(* CODESYS project SNDLTN_JSON.library
   Description: Library to convert and handle JSON data.
   Company: Sandolution
   Version: 1.2.200525
   Title: SNDLTN_JSON
   Author: S. Verbeek

Project tree, tasks and I/O mapping:
  libraries: StringUtils, * (System)
  Constants/
    global variables JSON_Properties
    global variables JSON_Constants
  Enums/
    data type JSON_eConversionType
    data type JSON_eError
  Function Blocks/
    function block JSON_Parser [ST]
    function block JSON_GetSingleValue [ST]
    function block JSON_GetMultiValue [ST]
  Functions/
  Structs/
  Variables/
  program ChangeLog [ST]
*)

// Enums/JSON_eConversionType
{attribute 'qualified_only'}
TYPE JSON_eConversionType :
(
	None := 0,				//NO CONVERSION
	Boolean,				//BOOL
	Integer,				//INT
	UnsignedInteger,		//UINT
	DoubleInteger,			//DINT
	UnsignedDoubleInteger,	//UDINT
	FloatingPoint,			//REAL
	DateAndTime,			//DT
	TimeOfDay				//TOD
);
END_TYPE

// Enums/JSON_eError
{attribute 'qualified_only'}
TYPE JSON_eError :
(
	NoError 				:= 0,
	//3000-3999 : JSON ERRORS
	PropertiesArrayToSmall 	:= 3000,	//JSON Parser output array to small
	PropertySizeToSmall 	:= 3001		//JSON Size to small
);
END_TYPE

// Constants/JSON_Properties
{attribute 'qualified_only'}
VAR_GLOBAL CONSTANT
	uiJSONMaxInputSize			:UINT := 4096;
	uiJSONMaxProperties			:UINT := 128;
	uiJSONMaxPropertySize		:UINT := 256;
	uiJSONMaxInputMultiValue	:UINT := 32;

END_VAR

// Constants/JSON_Constants
{attribute 'qualified_only'}
{attribute 'conditionalshow'}
VAR_GLOBAL
	sLineBreak					:STRING(1) := '$N';
	sColom						:STRING(3) := ' : ';
	sComma						:STRING(1) := ',';
	sQuotationMark				:STRING(1) := '"';
	sEnumerationBegin			:STRING(1) := '[';
	sEnumerationEnd				:STRING(1) := ']';
	sAccoladeBegin				:STRING(1) := '{';
	sAccoladeEnd				:STRING(1) := '}';
END_VAR

// Function Blocks/JSON_Parser
{attribute 'conditionalshow_all_locals'}
FUNCTION_BLOCK JSON_Parser
VAR_INPUT
	xResetError				:BOOL;
	sContent				:STRING(JSON_Properties.uiJSONMaxInputSize);
END_VAR
VAR_OUTPUT
	xError					:BOOL;
	eErrorID				:JSON_eError;
	
	//Double array: property/value
	asProperties			:ARRAY[0..1,0..JSON_Properties.uiJSONMaxProperties] OF STRING (JSON_Properties.uiJSONMaxPropertySize);
	uiPropertyCount			:UINT;
	xEnumerationPresent		:BOOL;	//Data contains one or more enumerations of multiple elements
	uiEnumerationIndex		:UINT;	//Start of FIRST enumeration
END_VAR
VAR
	//Store input
	sContent_int			:STRING(JSON_Properties.uiJSONMaxInputSize);
	
	//Input
	psContent				:POINTER TO STRING(JSON_Properties.uiJSONMaxInputSize);
	
	//Get total property line
	sProperty				:STRING(JSON_Properties.uiJSONMaxPropertySize);
	psProperty				:POINTER TO STRING(JSON_Properties.uiJSONMaxPropertySize);
	
	//Search for char (newline / comma / colon)
	sSearch					:STRING(4) := JSON_Constants.sLineBreak;	//Search for line end char
	psSearch				:POINTER TO STRING(4);
	
	//Output
	psProperties			:POINTER TO STRING (JSON_Properties.uiJSONMaxPropertySize);      	
	        
	//Helper            	
	diContentLength			:DINT;	//Length of content
	diPropertyLength		:DINT;	//Length of property
                	
	uiIndex					:UINT;
	
	iPosNewLine				:INT;
	iPosNewLine_Old			:INT;
	
	iPosColom				:INT;
	iPosQuotationMark_Begin	:ARRAY[0..1] OF INT;
	iPosQuotationMark_End	:ARRAY[0..1] OF INT;
	iPosQuotationMark_Loop	:INT;
	iPosComma				:INT;
	
	xOutput_Mem				:BOOL;	//Output written
END_VAR

//Get address and length
psContent := ADR(sContent);
psProperty := ADR(sProperty);
psSearch := ADR(sSearch);
diContentLength := StrLenA(psContent);

//Reset vars
iPosNewLine_Old := -1;	
xOutput_Mem := FALSE;

//Reset outputs
xEnumerationPresent := FALSE;

//Reset error
IF xResetError THEN
	xError := FALSE;
	eErrorID := JSON_eError.NoError;
END_IF

//Loop properties when input changed
IF sContent <> sContent_int THEN
	sContent_int := sContent;

	//Fill output array
	FOR uiIndex := 0 TO JSON_Properties.uiJSONMaxProperties DO
		
		//****************************************************GET PROPERTY FROM STRING (LINE BREAK)
		//Find pos of line break
		sSearch := JSON_Constants.sLineBreak;
		iPosNewLine := StrFindA(psContent, psSearch, TO_UINT(iPosNewLine_Old+1));
		
		IF iPosNewLine > 0 THEN
			
			//Get line at start of string
			IF uiIndex = 0 THEN	
				//Check if content fits the output
				IF (iPosNewLine-1) <= TO_INT(JSON_Properties.uiJSONMaxPropertySize) THEN
					StrMidA(psContent, JSON_Properties.uiJSONMaxInputSize, (iPosNewLine), 1, psProperty, JSON_Properties.uiJSONMaxPropertySize);
				ELSE
					xError := TRUE;
					eErrorID := JSON_eError.PropertySizeToSmall;
					EXIT;
				END_IF
			//Get line after first line
			ELSE	
				//Check if content fits the output
				IF (iPosNewLine-iPosNewLine_Old) <= TO_INT(JSON_Properties.uiJSONMaxPropertySize) THEN
					StrMidA(psContent, JSON_Properties.uiJSONMaxInputSize, (iPosNewLine-iPosNewLine_Old), (iPosNewLine_Old+1), psProperty, JSON_Properties.uiJSONMaxPropertySize);
				ELSE
					xError := TRUE;
					eErrorID := JSON_eError.PropertySizeToSmall;
					EXIT;
				END_IF
			END_IF
			
			//Store var for next find instruction
			iPosNewLine_Old := iPosNewLine;
			
			//****************************************************FIND COLOM IN PROPERTY
			sSearch := JSON_Constants.sColom;
			iPosColom := StrFindA(psProperty, psSearch, 0);
			
			//Column found	
			IF iPosColom > 0 THEN
			
				//****************************************************FIND NAME AND VALUE
				sSearch := JSON_Constants.sQuotationMark;
				//Name
				iPosQuotationMark_Begin[0] := StrFindA(psProperty, psSearch, 0);
				iPosQuotationMark_End[0] := StrFindA(psProperty, psSearch, TO_UINT(iPosQuotationMark_Begin[0]+1));
				
				//Value
				iPosQuotationMark_Begin[1] := StrFindA(psProperty, psSearch, TO_UINT(iPosColom));	//Search after colom
				
				//Start at back of string and work forwards to find latest one, enabling quotation marks in the value
				iPosQuotationMark_End[1] := 0;
				FOR iPosQuotationMark_Loop := TO_INT(StrLenA(psProperty)-1) TO (iPosQuotationMark_Begin[1]+1) BY -1 DO
					iPosQuotationMark_End[1] := StrFindA(psProperty, psSearch, TO_UINT(iPosQuotationMark_Loop));
					//Break if occurance is found
					IF iPosQuotationMark_End[1] <> 0 THEN 
						EXIT; 
					END_IF
				END_FOR
				
				//****************************************************EXTRACT NAME AND VALUE
				//Name
				psProperties := ADR(asProperties[0,uiIndex]);
				IF (iPosQuotationMark_End[0]-iPosQuotationMark_Begin[0]-1) <= TO_INT(JSON_Properties.uiJSONMaxPropertySize) THEN 
					StrMidA(psProperty, JSON_Properties.uiJSONMaxInputSize, (iPosQuotationMark_End[0]-iPosQuotationMark_Begin[0]-1), (iPosQuotationMark_Begin[0]+1), psProperties, JSON_Properties.uiJSONMaxPropertySize);
					StrTrimA(psProperties);	//Remove spaces
				ELSE
					xError := TRUE;
					eErrorID := JSON_eError.PropertySizeToSmall;
					EXIT;
				END_IF
				
				//Value with quotation marks
				psProperties := ADR(asProperties[1,uiIndex]);
				//Check if content fits the output
				IF iPosQuotationMark_Begin[1] > 0 AND iPosQuotationMark_End[1] > 0 THEN
					StrMidA(psProperty, JSON_Properties.uiJSONMaxInputSize, (iPosQuotationMark_End[1]-iPosQuotationMark_Begin[1]-1), (iPosQuotationMark_Begin[1]+1), psProperties, JSON_Properties.uiJSONMaxPropertySize);
					StrTrimA(psProperties);	//Remove spaces			
				
				//Value without quotation marks
				ELSE
					//Search for ending comma
					sSearch := JSON_Constants.sComma;
					iPosComma := StrFindA(psProperty, psSearch, 0);
					diPropertyLength := StrLenA(psProperty);
					//Extract to end of line minus one
					IF iPosComma > 0 THEN
						StrMidA(psProperty, JSON_Properties.uiJSONMaxInputSize, (TO_INT(diPropertyLength)-iPosColom-3-1), (iPosColom+3), psProperties, JSON_Properties.uiJSONMaxPropertySize);	//3> Search argument is ' : "  //1> skip comma
						StrTrimA(psProperties);	//Remove spaces
					//Extract to end of line
					ELSE		
						StrMidA(psProperty, JSON_Properties.uiJSONMaxInputSize, (TO_INT(diPropertyLength)-iPosColom-3), (iPosColom+3), psProperties, JSON_Properties.uiJSONMaxPropertySize);	//3> Search is ' : "
						StrTrimA(psProperties);	//Remove spaces
					END_IF
				END_IF
				
				//Check if there is more data then array size
				IF diContentLength > iPosQuotationMark_End[1] AND uiIndex = JSON_Properties.uiJSONMaxProperties THEN
					xError := TRUE;
					eErrorID := JSON_eError.PropertiesArrayToSmall;
				END_IF
				
				//Check if enumeration is present in array (for e.g. multiple instances of same object)
				//Find function is not used here as value can also be in a value
				IF NOT xEnumerationPresent 
				AND (asProperties[0,uiIndex] = JSON_Constants.sEnumerationBegin OR asProperties[0,uiIndex] = JSON_Constants.sEnumerationEnd
				OR asProperties[1,uiIndex] = JSON_Constants.sEnumerationBegin OR asProperties[1,uiIndex] = JSON_Constants.sEnumerationEnd) THEN
					xEnumerationPresent := TRUE;
					uiEnumerationIndex := uiIndex; 
				END_IF
			
			//No column found > no name+value but different charachter
			ELSE
				//Remove line break
				diPropertyLength := StrLenA(psProperty);
				StrMidA(psProperty, JSON_Properties.uiJSONMaxInputSize, TO_INT(diPropertyLength-1), 1, psProperty, JSON_Properties.uiJSONMaxPropertySize);
				
				//Transfer
				StrTrimA(psProperty);	//Remove spaces
				asProperties[0,uiIndex] := psProperty^;
				asProperties[1,uiIndex] := '';
				
				//Check if enumeration is present in array (for e.g. multiple instances of same object)
				//Find function is not used here as value can also be in a value
				IF NOT xEnumerationPresent 
				AND (asProperties[0,uiIndex] = JSON_Constants.sEnumerationBegin OR asProperties[0,uiIndex] = JSON_Constants.sEnumerationEnd) THEN
					xEnumerationPresent := TRUE;
					uiEnumerationIndex := uiIndex; 
				END_IF
				
			END_IF
			
		//Get latest part of string(should be closing accolade)
		ELSIF iPosNewLine_Old < diContentLength THEN
			IF (TO_INT(diContentLength)-iPosNewLine_Old) <= TO_INT(JSON_Properties.uiJSONMaxPropertySize) THEN
				StrMidA(psContent, JSON_Properties.uiJSONMaxInputSize, (TO_INT(diContentLength)-iPosNewLine_Old-1), iPosNewLine_Old+1, psProperty, JSON_Properties.uiJSONMaxPropertySize);
				StrTrimA(psProperty);	//Remove spaces
			ELSE
				xError := TRUE;
				eErrorID := JSON_eError.PropertySizeToSmall;
				EXIT;
			END_IF
			
			//Transfer data
			asProperties[0,uiIndex] := psProperty^;
			asProperties[1,uiIndex] := '';
			iPosNewLine_Old := TO_INT(diContentLength);
		
		//Closing function
		ELSIF iPosNewLine <= 0 AND iPosNewLine_Old = diContentLength THEN
			
			//Output property count
			IF NOT xOutput_Mem THEN
				xOutput_Mem := TRUE;
				uiPropertyCount := uiIndex;
			END_IF
			
			//Empty array after closing
			IF uiIndex >= uiPropertyCount THEN 
				asProperties[0,uiIndex] := '';
				asProperties[1,uiIndex] := '';
			END_IF
			
		END_IF
		
	END_FOR
END_IF

END_FUNCTION_BLOCK

// Function Blocks/JSON_GetSingleValue
{attribute 'conditionalshow_all_locals'}
FUNCTION_BLOCK JSON_GetSingleValue
VAR_INPUT
	pasProperties		:POINTER TO ARRAY[0..1,0..JSON_Properties.uiJSONMaxProperties] OF STRING(JSON_Properties.uiJSONMaxPropertySize);		//Pointer to output array
	sPropertyName		:STRING(JSON_Properties.uiJSONMaxPropertySize);
	eConversionType		:JSON_eConversionType;
END_VAR
VAR_OUTPUT
	xMatchFound			:BOOL;
	sPropertyValue		:STRING(JSON_Properties.uiJSONMaxPropertySize);		//Always loaded with value
	xPropertyValue		:BOOL;
	iPropertyValue		:INT;
	uiPropertyValue		:UINT;
	diPropertyValue		:DINT;
	udiPropertyValue	:UDINT;
	rPropertyValue		:REAL;
	dtPropertyValue		:DATE_AND_TIME;
	todPropertyValue	:TOD;
END_VAR
VAR
	iIndex				:INT;
	psPropertyValue		:POINTER TO STRING(JSON_Properties.uiJSONMaxPropertySize);
	sSearch				:STRING(8);
	psSearch			:POINTER TO STRING(8);
	iFindResult			:INT;
	
	sReplace			:STRING(1) := '-';
	psReplace			:POINTER TO STRING(4);
	
	sDateTime			:STRING(JSON_Properties.uiJSONMaxPropertySize) := 'DT#';
	psDateTime			:POINTER TO STRING(JSON_Properties.uiJSONMaxPropertySize);
	
	sTimeOfDay			:STRING(JSON_Properties.uiJSONMaxPropertySize) := 'TOD#';
	psTimeOfDay			:POINTER TO STRING(JSON_Properties.uiJSONMaxPropertySize);
	sTimeOfDay_Seconds	:STRING(JSON_Properties.uiJSONMaxPropertySize) := ':00';
	psTimeOfDay_Seconds	:POINTER TO STRING(JSON_Properties.uiJSONMaxPropertySize);
	
	iLengthTOD			:INT;
END_VAR

//Reset values
xMatchFound := FALSE;	//Assume no match is found
sPropertyValue := '';
xPropertyValue := 0;
iPropertyValue := 0;
uiPropertyValue := 0;
diPropertyValue := 0;
udiPropertyValue := 0;
rPropertyValue := 0;
dtPropertyValue := DT#1970-1-1-0:0:0;
todPropertyValue := TOD#0:0:0;

//Get addresses
psPropertyValue := ADR(sPropertyValue);
psSearch := ADR(sSearch);
psReplace := ADR(sReplace);
psDateTime := ADR(sDateTime);
psTimeOfDay := ADR(sTimeOfDay);
psTimeOfDay_Seconds := ADR(sTimeOfDay_Seconds);

IF sPropertyName <> '' AND pasProperties <> 0 THEN	//Property name filled in and pointer is valid
	FOR iIndex := 0 TO TO_INT(JSON_Properties.uiJSONMaxProperties) DO
		IF pasProperties^[0,iIndex] = sPropertyName THEN
			sPropertyValue := pasProperties^[1,iIndex];
			xMatchFound := TRUE;
			EXIT;
		END_IF
	END_FOR
END_IF

IF xMatchFound THEN
	CASE eConversionType OF
		
		JSON_eConversionType.Boolean:
			xPropertyValue := TO_BOOL(sPropertyValue);
			
		JSON_eConversionType.Integer:
			iPropertyValue := TO_INT(sPropertyValue);
			
		JSON_eConversionType.UnsignedInteger:
			uiPropertyValue := TO_UINT(sPropertyValue);
			
		JSON_eConversionType.DoubleInteger:
			diPropertyValue := TO_DINT(sPropertyValue);
			
		JSON_eConversionType.UnsignedDoubleInteger:
			udiPropertyValue := TO_UDINT(sPropertyValue);
			
		JSON_eConversionType.FloatingPoint:
			rPropertyValue := TO_REAL(sPropertyValue);
			
		JSON_eConversionType.DateAndTime:
			//Load vars
			sSearch := ' ';
			sReplace := '-';
			sDateTime := 'DT#';
			
			//Search for space in string
			iFindResult := StrFindA(psPropertyValue, psSearch, 1);
			IF iFindResult > 0 AND sPropertyValue <> '' THEN
				StrReplaceA(psPropertyValue, JSON_Properties.uiJSONMaxPropertySize, psReplace, TO_INT(StrLenA(psPropertyValue)), 1, 1, iFindResult);
				StrConcatA(psPropertyValue, psDateTime, TO_INT(JSON_Properties.uiJSONMaxPropertySize));
				dtPropertyValue := TO_DT(sDateTime);
			//If no spaces, conclude that format is already right
			ELSE
				StrConcatA(psPropertyValue, psDateTime, TO_INT(JSON_Properties.uiJSONMaxPropertySize));
				dtPropertyValue := TO_DT(sDateTime);
			END_IF
			
		JSON_eConversionType.TimeOfDay:
			//Load type definer
			sTimeOfDay := 'TOD#';
			StrConcatA(psPropertyValue, psTimeOfDay, TO_INT(JSON_Properties.uiJSONMaxPropertySize));		
	
			//Check length of string
			iLengthTOD := TO_INT(StrLenA(psTimeOfDay));
			
			//Check if seconds should be added
			IF iLengthTOD <= 9 THEN		//TOD#07:31
				sTimeOfDay_Seconds := ':00';
				StrConcatA(psTimeOfDay_Seconds, psTimeOfDay, TO_INT(JSON_Properties.uiJSONMaxPropertySize));
			END_IF
			
			todPropertyValue := TO_TOD(sTimeOfDay);
			
	END_CASE
END_IF

END_FUNCTION_BLOCK

// ChangeLog
PROGRAM ChangeLog
VAR
END_VAR

//Library for parsing JSON data to an usable (double) array. Breaks single string by special characters as defined in the JSON standard.
//Also provides a funcion to retreive a property from the (double) array.

//V1.2 - May 2020
//Update to compiler version 3.5.14.40

//V1.1 - Jan 2019
//Added EXIT condition to single value FOR-loop.
//Changed conditionalshow attributes
//Changed some constants into properties
//Removed xBusy from parser

//V1.0 - Dec 2018:
//Implementation of function blocks.
//Limitations: cannot handle multiple repeating properties, always takes first entry.

END_PROGRAM

// Function Blocks/JSON_GetMultiValue
{attribute 'conditionalshow_all_locals'}
FUNCTION_BLOCK JSON_GetMultiValue
VAR_INPUT
	pasProperties		:POINTER TO ARRAY[0..1,0..JSON_Properties.uiJSONMaxProperties] OF STRING(JSON_Properties.uiJSONMaxPropertySize);		//Pointer to output of parser
	asPropertyName		:ARRAY[0..JSON_Properties.uiJSONMaxInputMultiValue] OF STRING(JSON_Properties.uiJSONMaxPropertySize);
	aeConversionType	:ARRAY[0..JSON_Properties.uiJSONMaxInputMultiValue] OF JSON_eConversionType;
END_VAR
VAR_OUTPUT
	axMatchFound		:ARRAY[0..JSON_Properties.uiJSONMaxInputMultiValue] OF BOOL;
	asPropertyValue		:ARRAY[0..JSON_Properties.uiJSONMaxInputMultiValue] OF STRING(JSON_Properties.uiJSONMaxPropertySize);		//Always loaded with value
	axPropertyValue		:ARRAY[0..JSON_Properties.uiJSONMaxInputMultiValue] OF BOOL;
	aiPropertyValue		:ARRAY[0..JSON_Properties.uiJSONMaxInputMultiValue] OF INT;
	auiPropertyValue	:ARRAY[0..JSON_Properties.uiJSONMaxInputMultiValue] OF UINT;
	adiPropertyValue	:ARRAY[0..JSON_Properties.uiJSONMaxInputMultiValue] OF DINT;
	audiPropertyValue	:ARRAY[0..JSON_Properties.uiJSONMaxInputMultiValue] OF UDINT;
	arPropertyValue		:ARRAY[0..JSON_Properties.uiJSONMaxInputMultiValue] OF REAL;
	adtPropertyValue	:ARRAY[0..JSON_Properties.uiJSONMaxInputMultiValue] OF DATE_AND_TIME;
	atodPropertyValue	:ARRAY[0..JSON_Properties.uiJSONMaxInputMultiValue] OF TOD;
END_VAR
VAR
	aFB_GetSingleValue	:ARRAY[0..JSON_Properties.uiJSONMaxInputMultiValue] OF JSON_GetSingleValue;
	iForLoop			:INT;
END_VAR

//Call all FBs with settings

FOR iForLoop := 0 TO TO_INT(JSON_Properties.uiJSONMaxInputMultiValue) DO
	aFB_GetSingleValue[iForLoop](
	pasProperties := pasProperties, 
	sPropertyName:= asPropertyName[iForLoop], 
	eConversionType:= aeConversionType[iForLoop], 
	xMatchFound=> axMatchFound[iForLoop], 
	sPropertyValue=> asPropertyValue[iForLoop], 
	xPropertyValue=> axPropertyValue[iForLoop], 
	iPropertyValue=> aiPropertyValue[iForLoop], 
	uiPropertyValue=> auiPropertyValue[iForLoop], 
	diPropertyValue=> adiPropertyValue[iForLoop], 
	udiPropertyValue=> audiPropertyValue[iForLoop], 
	rPropertyValue=> arPropertyValue[iForLoop], 
	dtPropertyValue=> adtPropertyValue[iForLoop], 
	todPropertyValue=> atodPropertyValue[iForLoop]);
END_FOR

END_FUNCTION_BLOCK
